PROGRAM Pelletizer_Control
VAR
	Pelletizer_Lower_Status_Byte : UINT;
	
	Status_BitMask : UINT := 65280;
	DigitalInputStatus: INT;
END_VAR

//Bit 15 is digital input 1 which is the pelletizer control relay. If both of these are ON, we are in a started state.
IF (GVL_Pelletizer.MyPelletizer.Feedroll_VFD.VFD_Digital_Input_Status.16 = TRUE) AND (GVL_Pelletizer.MyPelletizer.Rotor_VFD.VFD_Digital_Input_Status.16 = TRUE) THEN
	GVL_Pelletizer.MyPelletizer.Pelletizer_Start := TRUE;
ELSE	
	GVL_Pelletizer.MyPelletizer.Pelletizer_Start := FALSE;
END_IF




//Fault Handling
GVL_Pelletizer.MyPelletizer.Feedroll_VFD.VFD_Fault := GVL_Pelletizer.MyPelletizer.Feedroll_VFD.VFD_Status_Word.3;
GVL_Pelletizer.MyPelletizer.Rotor_VFD.VFD_Fault := GVL_Pelletizer.MyPelletizer.Rotor_VFD.VFD_Status_Word.3;
//Overall Machine Fault if one or both drives faulted. 
IF (GVL_Pelletizer.MyPelletizer.Feedroll_VFD.VFD_Fault) OR (GVL_Pelletizer.MyPelletizer.Rotor_VFD.VFD_Fault) THEN
	GVL_Pelletizer.MyPelletizer.Pelletizer_Fault := TRUE;
ELSE
	GVL_Pelletizer.MyPelletizer.Pelletizer_Fault := FALSE;	
END_IF



//Reset faults
IF GVL_Pelletizer.MyPelletizer.Pelletizer_Fault_Reset THEN
	GVL_Pelletizer.MyPelletizer.Feedroll_VFD.VFD_Fault_Reset := TRUE;
	GVL_Pelletizer.MyPelletizer.Rotor_VFD.VFD_Fault_Reset := TRUE;
ELSE
	GVL_Pelletizer.MyPelletizer.Feedroll_VFD.VFD_Fault_Reset := FALSE;
	GVL_Pelletizer.MyPelletizer.Rotor_VFD.VFD_Fault_Reset := FALSE;
END_IF
//Set Reset
GVL_Pelletizer.MyPelletizer.Feedroll_VFD.VFD_Control_Word.7 := GVL_Pelletizer.MyPelletizer.Feedroll_VFD.VFD_Fault_reset;
GVL_Pelletizer.MyPelletizer.Rotor_VFD.VFD_Control_Word.7 := GVL_Pelletizer.MyPelletizer.Rotor_VFD.VFD_Fault_Reset;

END_PROGRAM

(* stored: Version 1.1.0.1, ProductVersion 3.1.4024.12
   POU Pelletizer_Control: Id {fab7e893-3672-4480-a2c7-2eaba39d3914}, SpecialFunc None *)
